// TIA Portal V20 export
DATA_BLOCK "T10 LANT"   // DB1193
{ S7_Optimized_Access := 'TRUE' }
AUTHOR : SAS
// stored: AutoNumber false, IsRetainMemResEnabled true, MemoryReserve 100, RetainMemoryReserve 100
   VAR RETAIN
      "Seq Status" : Struct
         ReadyToAuto : Bool;
         AutoON : Bool;
         WaitPiece : Bool;
         Stopped : Bool;
         "Step" : Struct
            Actual : Int;
            "-1" : Int;
            "-2" : Int;
            "-3" : Int;
            "-4" : Int;
            "-5" : Int;
            "-6" : Int;
            "-7" : Int;
            "-8" : Int;
            "-9" : Int;
            "Actual time" : Time_Of_Day;
            "-1 Time" : Time_Of_Day;
            "-2 Time" : Time_Of_Day;
            "-3 Time" : Time_Of_Day;
            "-4 Time" : Time_Of_Day;
            "-5 Time" : Time_Of_Day;
            "-6 Time" : Time_Of_Day;
            "-7 Time" : Time_Of_Day;
            "-8 Time" : Time_Of_Day;
            "-9 Time" : Time_Of_Day;
         END_STRUCT;
      END_STRUCT;
      Transitions : Struct
         Safe : Bool;   // Emergency
         Fault : Bool;   // Fault
         Auto : Bool;
         Manual : Bool;
         Semi_Auto : Bool;
         Pause : Bool;
         Stop : Bool;
         "Cycle start request" : Bool;
         "First Piece" : Bool;
         "Piece presence" : Bool;
         "Adjacent Machines" : Bool;
         "Adjacent Machines Repositioning" : Bool;   // Only for repositioning
         Init_Sequence : Bool;
         "Movement conditions 1" : Bool;   // Chain last position empty
         "Movement conditions 2" : Bool;
         "Movement conditions 3" : Bool;
         "Movement conditions 4" : Bool;
         "Reset Fault" : Bool;
         "Bypass ilock" : Bool;
      END_STRUCT;
      Memory : Struct
         "Piece presence" : Bool;   // Cumulative piece presence
         "Piece absence" : Bool;   // No sensor triggered
         Aux_PT_Start : Bool;   // Aux Prezenta Prima Pozitie Lant
         PT_Start : Bool;   // Prezenta Teava pe Pozitia Start Bancal
         TIME_OUT_BENCH : Bool;   // TimeOutBancal
         PT_END : Bool;   // Prezenta Teava Pozitie Stop Bancl
         MEM_PT_END : Bool;   // Memorie Teava Ultima Pozitie Lant
         TRK_PIPE_LAST : Bool;   // PIPE IN CHAIN LAST POSITION
         TRK_PIPE_IN : Bool;   // PIPE IN CHAIN RALL POSITION
         TRK_PIPE_Incet : Bool;   // ONE PIPE IN Incet POSITION
         Aux_PT_RALL : Bool;   // AUX Prezenta In Pozitie Slow
         PT_RALL : Bool;   // Prezenta Teava Incet Pozitie Bancal
         PIPE_TO_CHARGE : Bool;   // 1 pipe to charge
         C_PT : Bool;   // Cycle FILLING
         C_TO : Bool;   // Cycle Time out
         C_E : Bool;   // Cycle Empty
         C_F : Bool;   // Cycle Fast One pipe
         "Permanent Condition" : Bool;   // Permanent condition
         "Movement Fault" : Bool;   // Cumulative of Machine Fault condition
         "Local StopAuto" : Bool;   // Local StopAuto
         "Interlocks FW" : Bool;   // Interlocks for FORWARD
         "Interlocks BW" : Bool;   // Interlocks for BACKWARD
         "S8->S14" : Bool;   // From step 8 to step 14
         "S10->S14" : Bool;   // From step 10 to step 14
         "S12->S3" : Bool;   // From step 12 to step 3
         "S12->S8" : Bool;   // From step 12 to step 8
         "S12->S14" : Bool;   // From step 12 to step 14
         "S12->S16" : Bool;   // From step 12 to step 16
         Doi_Pasi : Bool;   // 0 = doi pasi done
         OS_CHAIN_STEP : Bool;   // Lant in 'Pas'
         "STEP" : Bool;   // Lant in 'Pas'
         "Lant T10" : Bool;   // Lant T10 (Pas)
         Lant_Pas_OK : Bool;   // Lant in Pas OK pentru Incarcare
         FW_ON : Bool;   // FORWARD ON
         BW_ON : Bool;   // BACKWARD ON
         CF_CHARGE_SPEED : Bool;   // FAST CYCLE: CHARGE SPEED REF.
         CF_DISCHARGE_SPEED : Bool;   // FAST CYCLE: DISCHARGE SPEED REF.
         CF_STANDBY_SPEED : Bool;   // FAST CYCLE: STAND-BY SPEED REF.
         CF_FAST_SPEED : Bool;   // FAST CYCLE: FAST SPEED REF.
         BENCH_EMPTY : Bool;   // Bancal Gol
         Dec_L1 : Bool;   // Decelerare L1
         Dec_L2 : Bool;   // Decelerare L2
         Dec_L3 : Bool;   // Decelerare L3
         Dec_L4 : Bool;   // Decelerare L4
         Dec_L5 : Bool;   // Decelerare L5
         Pas_Decel_Lant_T10 : Bool;   // Pas Decel Lant T10
         Stop_L1 : Bool;   // Stop L1
         Stop_L2 : Bool;   // Stop L2
         Stop_L3 : Bool;   // Stop L3
         Stop_L4 : Bool;   // Stop L4
         Stop_L5 : Bool;   // Stop L5
         Pas_Stop_Lant_T10 : Bool;   // Pas Stop Lant T10
         Aux_Oprire_Pas : Bool;   // Aux Oprire Lant In Pas In Mod Manual
         Frana : Bool;   // Frana
         Aux_CMD_Frana : Bool;   // 1 = CMD Decuplata
         COUNT_STEP : Int;   // Numar Pas Lant
         PASI : Int;   // Lant T10 Pasi
         SPEED_FW_AUTO_ROLL_MIN : Real;   // Viteza Teava 'Inainte' AUTO [ROLL\MINUTE]
         SPEED_FW_AUTO_RPM : Real;   // Viteza Teava 'Inainte' AUTO [RPM]
         SPEED_FW_AUTO_HZ : Real;   // Viteza Teava 'Inainte' AUTO [HZ*10]
         SPEED_OPERATIVE : Real;   // Viteza Operativa Teava [HZ*10]
         ROST_SPEED_OPERATIVE : Real;   // Referinta Viteza [HZ*10]
      END_STRUCT;
   END_VAR
BEGIN
END_DATA_BLOCK
